// TIA Portal V20 export
DATA_BLOCK "OEM_CITI_Logic_Setup"   // DB5800
// stored: MemoryReserve 0, Namespace CITI_Logic
   VAR
      OEM : Array[0..29] of "CITI_Logic.OEM_Data";
   END_VAR
BEGIN
END_DATA_BLOCK
